// TIA Portal V17 export
// export: Created 2022-07-20T07:02:39.8085966Z, ExportSetting WithDefaults, DisplayName Totally Integrated Automation Portal, DisplayVersion V17, DisplayName TIA Portal Openness, DisplayVersion V17, DisplayName TIA Portal Version Control Interface, DisplayVersion V17, DisplayName SINAMICS Startdrive Advanced, DisplayVersion V17, DisplayName SINAMICS Startdrive G130, G150, S120, S150, SINAMICS MV, S210, DisplayVersion V17, DisplayName SINAMICS Startdrive G110M, G120, G120C, G120D, G120P, G115D, DisplayVersion V17, DisplayName STEP 7 Professional, DisplayVersion V17, DisplayName STEP 7 Safety, DisplayVersion V17, DisplayName WinCC Advanced, DisplayVersion V17
VAR_GLOBAL   // PLC tag table "LCamHdl_ConfigConstants"
END_VAR
VAR_GLOBAL CONSTANT   // user constants
   LCAMHDL_DELETE_NO_DATA : DInt := 0;
   LCAMHDL_DELETE_DATA_UNTIL_FIRST_INVALID_DATA_FOUND : DInt := 1;
   LCAMHDL_DELETE_ALL_DATA : DInt := 2;
END_VAR
